// TIA Portal V20 export
TYPE "HMI_IF_OverView_Unit_UDT"
// stored: Access Published
   STRUCT
      State : Struct
         Communication : SInt;
         Mode : SInt;
         State : SInt;
         Emergency : SInt;
      END_STRUCT;
      "Link&Unlink" : Struct
         Em0 : Bool;
         Em1 : Bool;
         Em2 : Bool;
         Em3 : Bool;
         Em4 : Bool;
         Em5 : Bool;
         Em6 : Bool;
         Em7 : Bool;
         Em8 : Bool;
         Em9 : Bool;
         Em10 : Bool;
         Em11 : Bool;
         Em12 : Bool;
         Em13 : Bool;
         Em14 : Bool;
         Em15 : Bool;
      END_STRUCT;
      Production : Struct
         "Total Input Quantity" : DInt;
         "Remain Count" : DInt;
         "Processed Count" : DInt;
         "NG Count" : DInt;
      END_STRUCT;
   END_STRUCT;
END_TYPE
